VAR_GLOBAL
	//HOMS M1
	HOMS1_Pitch	    :	HOMS_PitchMechanism := (ReqPosLimHi:=0.13, ReqPosLimLo:=-0.08);
	HOMS1_YGantry	:	HOMS_Gantry;
	HOMS1_XGantry	:	HOMS_Gantry;
	HOMS1_Bender	:	ST_HOMSStepper;

	//HOMS M2
	HOMS2_Pitch	    : HOMS_PitchMechanism := (ReqPosLimHi:=0.09, ReqPosLimLo:=-0.15);
	HOMS2_YGantry	: HOMS_Gantry;
	HOMS2_XGantry	: HOMS_Gantry;
	
	
END_VAR

(* stored: Version 1.1.0.1, ProductVersion 3.1.4020.12
   GVL GVL_Devices: Id {cb7cf638-cc80-4f58-a532-470704faedf8} *)
